# B&R Automation Studio project ubiquitous-potato
Automation Studio 4.5.2.102

## Configuration Config1

### Task classes (Cpu.sw)
```
Cyclic#1:
  Program <- Program.prg
Binaries: udbdef, TCData, sysconf, Role, User, iomap, ashwd, asfw, arconfig, ashwac
Libraries: Library
```

### Hardware
```
4PP065_0351_P74 : 4PP065.0351-P74 v1.0.4.0
  Connector IF5:
    ActivateDevice = 1
    Mode = Manual
    InternetAddress = 10.0.1.10
    SubnetMask = 255.255.255.0
  ConfigurationID = labBR
  KeyMappingFile = VC\4PP065_0351_P74.dis
```

## Logical view

### Library Logical/Libraries/Library (ANSIC)

#### Library.fun - Exported functions and function blocks
```iecst
{REDUND_ERROR} FUNCTION_BLOCK FB_Motor (*TODO: Add your comment here*) (*$GROUP=User,$CAT=User,$GROUPICON=User.png,$CATICON=User.png*)
	VAR_INPUT
		u : {REDUND_UNREPLICABLE} REAL;
	END_VAR
	VAR_OUTPUT
		w : {REDUND_UNREPLICABLE} REAL;
		phi : {REDUND_UNREPLICABLE} REAL;
	END_VAR
	VAR
		integrator : {REDUND_UNREPLICABLE} FB_Integrator;
		Tm : {REDUND_UNREPLICABLE} REAL;
		ke : {REDUND_UNREPLICABLE} REAL;
		dt : {REDUND_UNREPLICABLE} REAL;
		motor_integrator : FB_Integrator;
		sensor_integrator : FB_Integrator;
	END_VAR
END_FUNCTION_BLOCK

{REDUND_ERROR} FUNCTION_BLOCK FB_Integrator (*TODO: Add your comment here*) (*$GROUP=User,$CAT=User,$GROUPICON=User.png,$CATICON=User.png*)
	VAR_INPUT
		in : {REDUND_UNREPLICABLE} REAL;
	END_VAR
	VAR_OUTPUT
		out : {REDUND_UNREPLICABLE} REAL;
	END_VAR
	VAR
		dt : {REDUND_UNREPLICABLE} REAL;
	END_VAR
	VAR_OUTPUT
		state : REAL;
	END_VAR
END_FUNCTION_BLOCK

{REDUND_ERROR} {REDUND_UNREPLICABLE} FUNCTION_BLOCK FB_Regulator (*TODO: Add your comment here*) (*$GROUP=User,$CAT=User,$GROUPICON=User.png,$CATICON=User.png*)
	VAR_INPUT
		e : {REDUND_UNREPLICABLE} REAL;
	END_VAR
	VAR_OUTPUT
		u : {REDUND_UNREPLICABLE} REAL;
	END_VAR
	VAR
		k_p : {REDUND_UNREPLICABLE} REAL;
		k_i : {REDUND_UNREPLICABLE} REAL;
		integrator : {REDUND_UNREPLICABLE} FB_Integrator;
		iyOld : {REDUND_UNREPLICABLE} REAL;
		max_abs_value : {REDUND_UNREPLICABLE} REAL;
		dt : {REDUND_UNREPLICABLE} REAL;
	END_VAR
END_FUNCTION_BLOCK
```

#### FB_Motor.c
```c
#include <bur/plctypes.h>
#ifdef __cplusplus
	extern "C"
	{
#endif
	#include "Library.h"
#ifdef __cplusplus
	};
#endif
/* MOTOR */
void FB_Motor(struct FB_Motor* inst)
{
    REAL b1 = inst->u * (1/inst->ke) - inst->w;
    REAL b2 = b1/ inst->Tm;

    inst->motor_integrator.in = b2;
    FB_Integrator(&inst->motor_integrator);

    inst->w = inst->motor_integrator.out;

    inst->sensor_integrator.in = inst->w;
    FB_Integrator(&inst->sensor_integrator);

    inst->phi = inst->sensor_integrator.out ;

}
```

#### FB_Regulator.c
```c
#include <bur/plctypes.h>
#ifdef __cplusplus
	extern "C"
	{
#endif
	#include "Library.h"
#ifdef __cplusplus
	};
#endif
/* REGULATOR */
void FB_Regulator(struct FB_Regulator* inst)
{
    REAL p_part = inst->e * inst->k_p;

    REAL i_part = inst->e * inst->k_i;

    inst->integrator.in = i_part;

    FB_Integrator(&inst->integrator);

    i_part = inst->integrator.out;

    REAL total_output = p_part + i_part;

    if (total_output > inst->max_abs_value)
    {
        inst->u = inst->max_abs_value;
        inst->integrator.out = inst->max_abs_value - p_part;

    } else if (total_output < -inst->max_abs_value)
    {
        inst->u = -inst->max_abs_value;
        inst->integrator.out = -inst->max_abs_value - p_part;
    } else
    {
        inst->u = total_output;

    }
    inst->iyOld = i_part;
}
```

#### FB_Integrator.c
```c
#include <bur/plctypes.h>
#ifdef __cplusplus
	extern "C"
	{
#endif
	#include "Library.h"
#ifdef __cplusplus
	};
#endif
/* INTEGRATOR */
void FB_Integrator(struct FB_Integrator* inst)
{
    inst->dt= 0.01;

    inst->out = inst->dt * inst->in + inst->state;
    inst->state = inst->out;
}
```

### Program Logical/Program

#### Variables.var
```iecst
VAR
	speed_in_rad : REAL;
	enable : USINT;
	speed : UINT;
	counter : UDINT;
	fb_controller : FB_Regulator;
	fb_motor2 : FB_Motor;
	fb_motor : FB_Motor;
END_VAR
```

#### Main.c
```c
#include <bur/plctypes.h>

#ifdef _DEFAULT_INCLUDES
	#include <AsDefault.h>
#endif

void _INIT ProgramInit(void)
{
    enable = 1;
    counter = 0;
    speed = 0;
	speed_in_rad = 0;

    fb_motor.dt=0.01;
    fb_motor.ke=2.65;
    fb_motor.Tm=0.05;

    fb_motor2.dt = 0.01;
    fb_motor2.ke = 2.65;
    fb_motor2.Tm = 0.05;

    fb_controller.dt=0.01;
    fb_controller.k_p = (fb_motor.ke* fb_motor.Tm) / 0.02;
    fb_controller.k_i = fb_motor.ke / 0.02;
    fb_controller.max_abs_value=24;
}

void _CYCLIC ProgramCyclic(void)
{
    REAL PI = 3.141592653589793;
    REAL desired_w = speed * 2.0 * PI / 60.0;
	speed_in_rad = desired_w;

    if (enable == 1){
        counter += 1;
        if ((counter >= 500 ) && (counter <= 1000)) speed = 70;
        else speed = 0;
    }
    else speed = 0;

    fb_controller.e = desired_w - fb_motor.w;
    FB_Regulator(&fb_controller);
	fb_motor.u = fb_controller.u;

    fb_motor2.u = desired_w * fb_motor2.ke;

    FB_Motor(&fb_motor);
    FB_Motor(&fb_motor2);

}

void _EXIT ProgramExit(void)
{

}
```

Listed in the project but not available here: Logical/Libraries/Library/Types.typ, Logical/Libraries/Library/Constants.var
